// TIA Portal V19 export
FUNCTION_BLOCK "F_Zone01_02_03_FB"   // FB114, F_LAD
TITLE = SAFETY ZONE 01 (DEC.ROTATION) / ZONE 02 (DECOILER 1) / ZONE 03 (DECOILER 2)
// stored: Access Published
   VAR
      D01 : "Door_FB";
      D02 : "Door_FB";
      D03 : "Door_FB";
      F_SafetyValve_DecoilersHorizRotation : "FDevice_Valve_FB";
      F_SafetyValve_Decoiler1 : "FDevice_Valve_FB";
      F_SafetyValve_Decoiler2 : "FDevice_Valve_FB";
      F_Contactor_HU_Decoilers_Motor : "FDevice_Contactor_FB";
      F_Sinamics_DecoilersTranslation : "FDevice_Sinamics_FB";
      F_Sinamics_Decoiler1 : "FDevice_Sinamics_FB";
      F_Sinamics_Decoiler2 : "FDevice_Sinamics_FB";
      Zone02_Close : Bool;
      Zone03_Close : Bool;
   END_VAR
   VAR CONSTANT
      DECOILER_S120_STOPPING_TIME : Time := t#2S;
   END_VAR
BEGIN

REGION Network 1: < < < < < < < < < < DOORS > > > > > > > > > >
END_REGION

REGION Network 2: Zone 01 - Entry enable
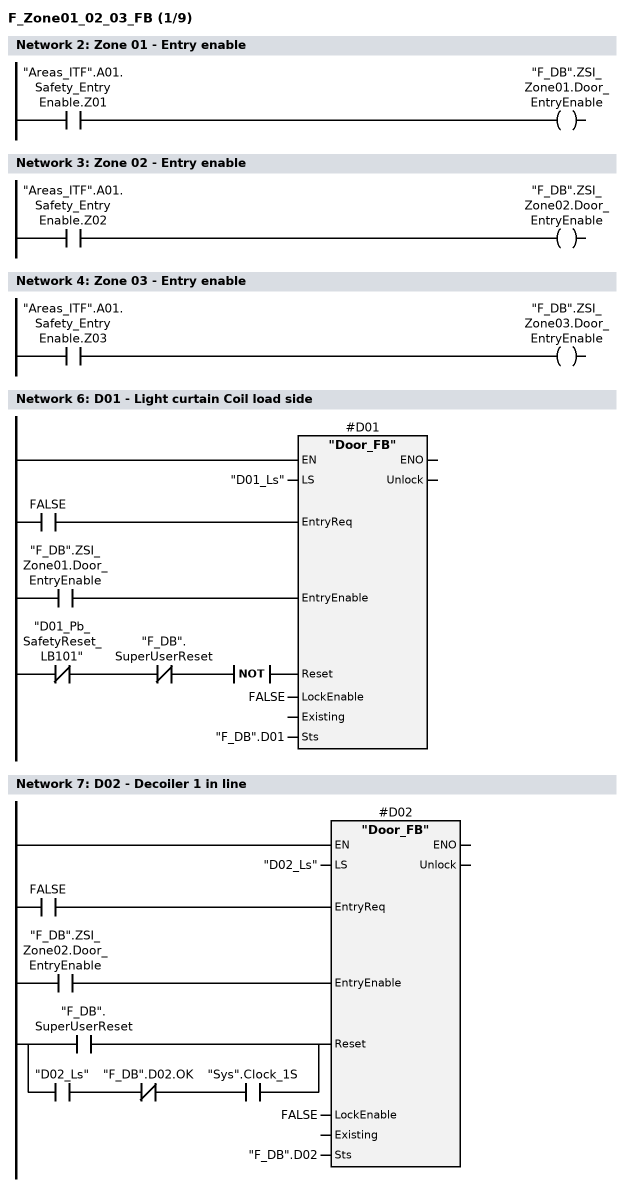
   RUNG wire#powerrail
      Contact( "Areas_ITF".A01.Safety_EntryEnable.Z01 )
      Coil( "F_DB".ZSI_Zone01.Door_EntryEnable )
   END_RUNG
   // the same network as SCL:
   "F_DB".ZSI_Zone01.Door_EntryEnable := "Areas_ITF".A01.Safety_EntryEnable.Z01;
END_REGION

REGION Network 3: Zone 02 - Entry enable
   RUNG wire#powerrail
      Contact( "Areas_ITF".A01.Safety_EntryEnable.Z02 )
      Coil( "F_DB".ZSI_Zone02.Door_EntryEnable )
   END_RUNG
   // the same network as SCL:
   "F_DB".ZSI_Zone02.Door_EntryEnable := "Areas_ITF".A01.Safety_EntryEnable.Z02;
END_REGION

REGION Network 4: Zone 03 - Entry enable
   RUNG wire#powerrail
      Contact( "Areas_ITF".A01.Safety_EntryEnable.Z03 )
      Coil( "F_DB".ZSI_Zone03.Door_EntryEnable )
   END_RUNG
   // the same network as SCL:
   "F_DB".ZSI_Zone03.Door_EntryEnable := "Areas_ITF".A01.Safety_EntryEnable.Z03;
END_REGION

REGION Network 5: >
END_REGION

REGION Network 6: D01 - Light curtain Coil load side
   RUNG wire#powerrail
      #D01(EntryReq := wire#w1, EntryEnable := wire#w2, Reset := wire#w3, LS := "D01_Ls", LockEnable := FALSE, Existing :=, Sts := "F_DB".D01, Unlock =>)
   END_RUNG
   RUNG wire#powerrail
      Contact( FALSE )
   END_RUNG wire#w1
   RUNG wire#powerrail
      Contact( "F_DB".ZSI_Zone01.Door_EntryEnable )
   END_RUNG wire#w2
   RUNG wire#powerrail
      I_Contact( "D01_Pb_SafetyReset_LB101" )
      I_Contact( "F_DB".SuperUserReset )
      Not()
   END_RUNG wire#w3
   // the same network as SCL:
   #D01(LS := "D01_Ls",   // "Door_FB"
        EntryReq := FALSE,
        EntryEnable := "F_DB".ZSI_Zone01.Door_EntryEnable,
        Reset := NOT (NOT "D01_Pb_SafetyReset_LB101" AND NOT "F_DB".SuperUserReset),
        LockEnable := FALSE,
        Sts := "F_DB".D01);
END_REGION

REGION Network 7: D02 - Decoiler 1 in line
   RUNG wire#powerrail
      #D02(EntryReq := wire#w1, EntryEnable := wire#w2, Reset := wire#w3, LS := "D02_Ls", LockEnable := FALSE, Existing :=, Sts := "F_DB".D02, Unlock =>)
   END_RUNG
   RUNG wire#powerrail
      Contact( FALSE )
   END_RUNG wire#w1
   RUNG wire#powerrail
      Contact( "F_DB".ZSI_Zone02.Door_EntryEnable )
   END_RUNG wire#w2
   RUNG wire#powerrail
      Contact( "F_DB".SuperUserReset )
   END_RUNG wire#w3
   RUNG wire#powerrail
      Contact( "D02_Ls" )
      I_Contact( "F_DB".D02.OK )
      Contact( "Sys".Clock_1S )
   END_RUNG wire#w3
   // the same network as SCL:
   #D02(LS := "D02_Ls",   // "Door_FB"
        EntryReq := FALSE,
        EntryEnable := "F_DB".ZSI_Zone02.Door_EntryEnable,
        Reset := "F_DB".SuperUserReset OR ("D02_Ls" AND NOT "F_DB".D02.OK AND "Sys".Clock_1S),
        LockEnable := FALSE,
        Sts := "F_DB".D02);
END_REGION

REGION Network 8: D03 - Decoiler 2 in line
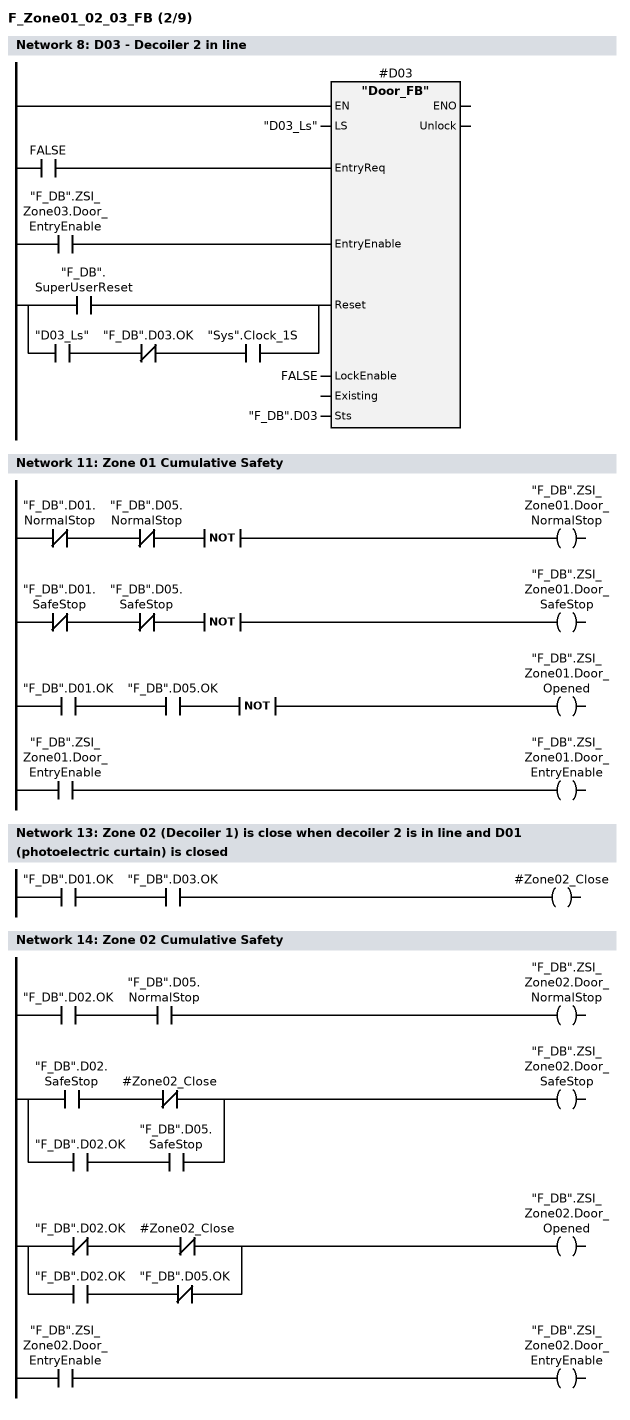
   RUNG wire#powerrail
      #D03(EntryReq := wire#w1, EntryEnable := wire#w2, Reset := wire#w3, LS := "D03_Ls", LockEnable := FALSE, Existing :=, Sts := "F_DB".D03, Unlock =>)
   END_RUNG
   RUNG wire#powerrail
      Contact( FALSE )
   END_RUNG wire#w1
   RUNG wire#powerrail
      Contact( "F_DB".ZSI_Zone03.Door_EntryEnable )
   END_RUNG wire#w2
   RUNG wire#powerrail
      Contact( "F_DB".SuperUserReset )
   END_RUNG wire#w3
   RUNG wire#powerrail
      Contact( "D03_Ls" )
      I_Contact( "F_DB".D03.OK )
      Contact( "Sys".Clock_1S )
   END_RUNG wire#w3
   // the same network as SCL:
   #D03(LS := "D03_Ls",   // "Door_FB"
        EntryReq := FALSE,
        EntryEnable := "F_DB".ZSI_Zone03.Door_EntryEnable,
        Reset := "F_DB".SuperUserReset OR ("D03_Ls" AND NOT "F_DB".D03.OK AND "Sys".Clock_1S),
        LockEnable := FALSE,
        Sts := "F_DB".D03);
END_REGION

REGION Network 9: >
END_REGION

REGION Network 10: < < < < < < < < < < ZONE SAFETY INTERFACE > > > > > > > > > >
END_REGION

REGION Network 11: Zone 01 Cumulative Safety
   RUNG wire#powerrail
      I_Contact( "F_DB".D01.NormalStop )
      I_Contact( "F_DB".D05.NormalStop )
      Not()
      Coil( "F_DB".ZSI_Zone01.Door_NormalStop )
   END_RUNG
   RUNG wire#powerrail
      I_Contact( "F_DB".D01.SafeStop )
      I_Contact( "F_DB".D05.SafeStop )
      Not()
      Coil( "F_DB".ZSI_Zone01.Door_SafeStop )
   END_RUNG
   RUNG wire#powerrail
      Contact( "F_DB".D01.OK )
      Contact( "F_DB".D05.OK )
      Not()
      Coil( "F_DB".ZSI_Zone01.Door_Opened )
   END_RUNG
   RUNG wire#powerrail
      Contact( "F_DB".ZSI_Zone01.Door_EntryEnable )
      Coil( "F_DB".ZSI_Zone01.Door_EntryEnable )
   END_RUNG
   // the same network as SCL:
   "F_DB".ZSI_Zone01.Door_NormalStop := NOT (NOT "F_DB".D01.NormalStop AND NOT "F_DB".D05.NormalStop);
   "F_DB".ZSI_Zone01.Door_SafeStop := NOT (NOT "F_DB".D01.SafeStop AND NOT "F_DB".D05.SafeStop);
   "F_DB".ZSI_Zone01.Door_Opened := NOT ("F_DB".D01.OK AND "F_DB".D05.OK);
   "F_DB".ZSI_Zone01.Door_EntryEnable := "F_DB".ZSI_Zone01.Door_EntryEnable;
END_REGION

REGION Network 12: >
END_REGION

REGION Network 13: Zone 02 (Decoiler 1) is close when decoiler 2 is in line and D01 (photoelectric curtain) is closed
   RUNG wire#powerrail
      Contact( "F_DB".D01.OK )
      Contact( "F_DB".D03.OK )
      Coil( #Zone02_Close )
   END_RUNG
   // the same network as SCL:
   #Zone02_Close := "F_DB".D01.OK AND "F_DB".D03.OK;
END_REGION

REGION Network 14: Zone 02 Cumulative Safety
   RUNG wire#powerrail
      Contact( "F_DB".D02.OK )
      Contact( "F_DB".D05.NormalStop )
      Coil( "F_DB".ZSI_Zone02.Door_NormalStop )
   END_RUNG
   RUNG wire#powerrail
      Contact( "F_DB".D02.SafeStop )
      I_Contact( #Zone02_Close )
      wire#w1
      Coil( "F_DB".ZSI_Zone02.Door_SafeStop )
   END_RUNG
   RUNG wire#powerrail
      Contact( "F_DB".D02.OK )
      Contact( "F_DB".D05.SafeStop )
   END_RUNG wire#w1
   RUNG wire#powerrail
      I_Contact( "F_DB".D02.OK )
      I_Contact( #Zone02_Close )
      wire#w2
      Coil( "F_DB".ZSI_Zone02.Door_Opened )
   END_RUNG
   RUNG wire#powerrail
      Contact( "F_DB".D02.OK )
      I_Contact( "F_DB".D05.OK )
   END_RUNG wire#w2
   RUNG wire#powerrail
      Contact( "F_DB".ZSI_Zone02.Door_EntryEnable )
      Coil( "F_DB".ZSI_Zone02.Door_EntryEnable )
   END_RUNG
   // the same network as SCL:
   "F_DB".ZSI_Zone02.Door_NormalStop := "F_DB".D02.OK AND "F_DB".D05.NormalStop;
   "F_DB".ZSI_Zone02.Door_SafeStop := ("F_DB".D02.SafeStop AND NOT #Zone02_Close) OR ("F_DB".D02.OK AND "F_DB".D05.SafeStop);
   "F_DB".ZSI_Zone02.Door_Opened := (NOT "F_DB".D02.OK AND NOT #Zone02_Close) OR ("F_DB".D02.OK AND NOT "F_DB".D05.OK);
   "F_DB".ZSI_Zone02.Door_EntryEnable := "F_DB".ZSI_Zone02.Door_EntryEnable;
END_REGION

REGION Network 15: >
END_REGION

REGION Network 16: Zone 03 (Decoiler 2) is close when decoiler 1 is in line and D01 (photoelectric curtain) is closed
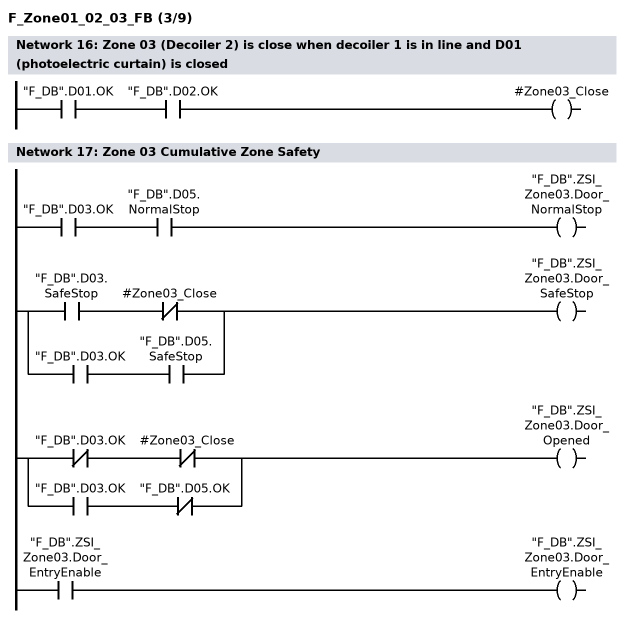
   RUNG wire#powerrail
      Contact( "F_DB".D01.OK )
      Contact( "F_DB".D02.OK )
      Coil( #Zone03_Close )
   END_RUNG
   // the same network as SCL:
   #Zone03_Close := "F_DB".D01.OK AND "F_DB".D02.OK;
END_REGION

REGION Network 17: Zone 03 Cumulative Zone Safety
   RUNG wire#powerrail
      Contact( "F_DB".D03.OK )
      Contact( "F_DB".D05.NormalStop )
      Coil( "F_DB".ZSI_Zone03.Door_NormalStop )
   END_RUNG
   RUNG wire#powerrail
      Contact( "F_DB".D03.SafeStop )
      I_Contact( #Zone03_Close )
      wire#w1
      Coil( "F_DB".ZSI_Zone03.Door_SafeStop )
   END_RUNG
   RUNG wire#powerrail
      Contact( "F_DB".D03.OK )
      Contact( "F_DB".D05.SafeStop )
   END_RUNG wire#w1
   RUNG wire#powerrail
      I_Contact( "F_DB".D03.OK )
      I_Contact( #Zone03_Close )
      wire#w2
      Coil( "F_DB".ZSI_Zone03.Door_Opened )
   END_RUNG
   RUNG wire#powerrail
      Contact( "F_DB".D03.OK )
      I_Contact( "F_DB".D05.OK )
   END_RUNG wire#w2
   RUNG wire#powerrail
      Contact( "F_DB".ZSI_Zone03.Door_EntryEnable )
      Coil( "F_DB".ZSI_Zone03.Door_EntryEnable )
   END_RUNG
   // the same network as SCL:
   "F_DB".ZSI_Zone03.Door_NormalStop := "F_DB".D03.OK AND "F_DB".D05.NormalStop;
   "F_DB".ZSI_Zone03.Door_SafeStop := ("F_DB".D03.SafeStop AND NOT #Zone03_Close) OR ("F_DB".D03.OK AND "F_DB".D05.SafeStop);
   "F_DB".ZSI_Zone03.Door_Opened := (NOT "F_DB".D03.OK AND NOT #Zone03_Close) OR ("F_DB".D03.OK AND NOT "F_DB".D05.OK);
   "F_DB".ZSI_Zone03.Door_EntryEnable := "F_DB".ZSI_Zone03.Door_EntryEnable;
END_REGION

REGION Network 18: >
END_REGION

REGION Network 19: < < < < < < < < < < DEVICES SAFETY VALVES > > > > > > > > > >
END_REGION

REGION Network 20: (Zone 01) HU Decoilers Safety Valve Decoilers Horizonatal Rotation
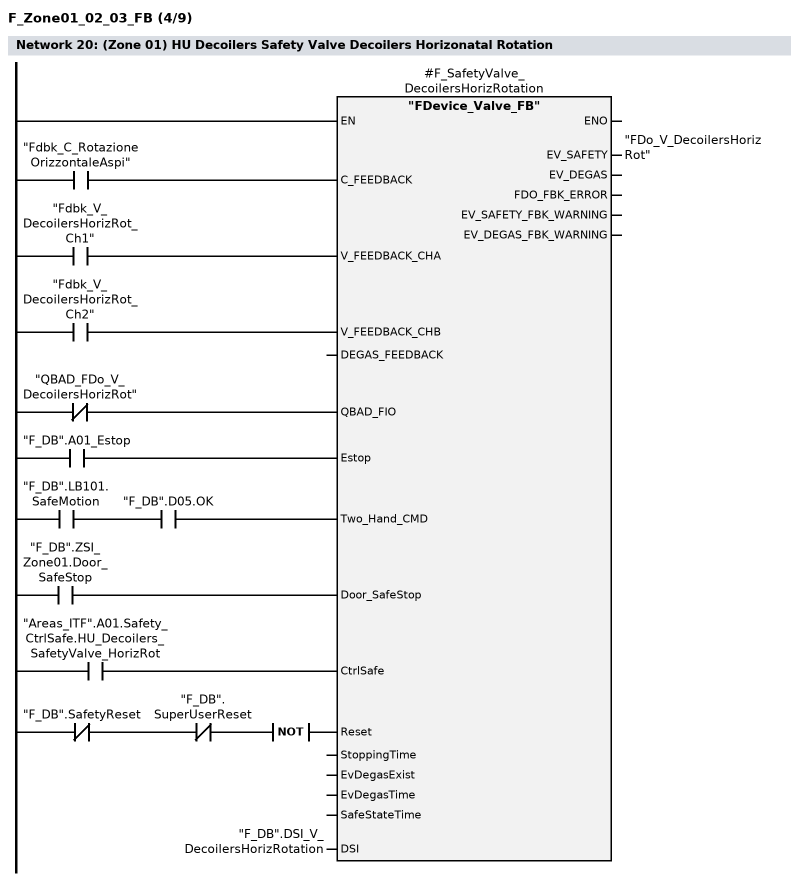
   RUNG wire#powerrail
      #F_SafetyValve_DecoilersHorizRotation(C_FEEDBACK := wire#w1, V_FEEDBACK_CHA := wire#w2, V_FEEDBACK_CHB := wire#w3, QBAD_FIO := wire#w4, Estop := wire#w5, Two_Hand_CMD := wire#w6, Door_SafeStop := wire#w7, CtrlSafe := wire#w8, Reset := wire#w9, DEGAS_FEEDBACK :=, StoppingTime :=, EvDegasExist :=, EvDegasTime :=, SafeStateTime :=, DSI := "F_DB".DSI_V_DecoilersHorizRotation, EV_SAFETY => "FDo_V_DecoilersHorizRot", EV_DEGAS =>, FDO_FBK_ERROR =>, EV_SAFETY_FBK_WARNING =>, EV_DEGAS_FBK_WARNING =>)
   END_RUNG
   RUNG wire#powerrail
      Contact( "Fdbk_C_RotazioneOrizzontaleAspi" )
   END_RUNG wire#w1
   RUNG wire#powerrail
      Contact( "Fdbk_V_DecoilersHorizRot_Ch1" )
   END_RUNG wire#w2
   RUNG wire#powerrail
      Contact( "Fdbk_V_DecoilersHorizRot_Ch2" )
   END_RUNG wire#w3
   RUNG wire#powerrail
      I_Contact( "QBAD_FDo_V_DecoilersHorizRot" )
   END_RUNG wire#w4
   RUNG wire#powerrail
      Contact( "F_DB".A01_Estop )
   END_RUNG wire#w5
   RUNG wire#powerrail
      Contact( "F_DB".LB101.SafeMotion )
      Contact( "F_DB".D05.OK )
   END_RUNG wire#w6
   RUNG wire#powerrail
      Contact( "F_DB".ZSI_Zone01.Door_SafeStop )
   END_RUNG wire#w7
   RUNG wire#powerrail
      Contact( "Areas_ITF".A01.Safety_CtrlSafe.HU_Decoilers_SafetyValve_HorizRot )
   END_RUNG wire#w8
   RUNG wire#powerrail
      I_Contact( "F_DB".SafetyReset )
      I_Contact( "F_DB".SuperUserReset )
      Not()
   END_RUNG wire#w9
   // the same network as SCL:
   #F_SafetyValve_DecoilersHorizRotation(C_FEEDBACK := "Fdbk_C_RotazioneOrizzontaleAspi",   // "FDevice_Valve_FB"
                           V_FEEDBACK_CHA := "Fdbk_V_DecoilersHorizRot_Ch1",
                           V_FEEDBACK_CHB := "Fdbk_V_DecoilersHorizRot_Ch2",
                           QBAD_FIO := NOT "QBAD_FDo_V_DecoilersHorizRot",
                           Estop := "F_DB".A01_Estop,
                           Two_Hand_CMD := "F_DB".LB101.SafeMotion AND "F_DB".D05.OK,
                           Door_SafeStop := "F_DB".ZSI_Zone01.Door_SafeStop,
                           CtrlSafe := "Areas_ITF".A01.Safety_CtrlSafe.HU_Decoilers_SafetyValve_HorizRot,
                           Reset := NOT (NOT "F_DB".SafetyReset AND NOT "F_DB".SuperUserReset),
                           DSI := "F_DB".DSI_V_DecoilersHorizRotation,
                           EV_SAFETY => "FDo_V_DecoilersHorizRot");
END_REGION

REGION Network 21: (Zone 02) HU Decoilers Safety Valve Decoiler 1
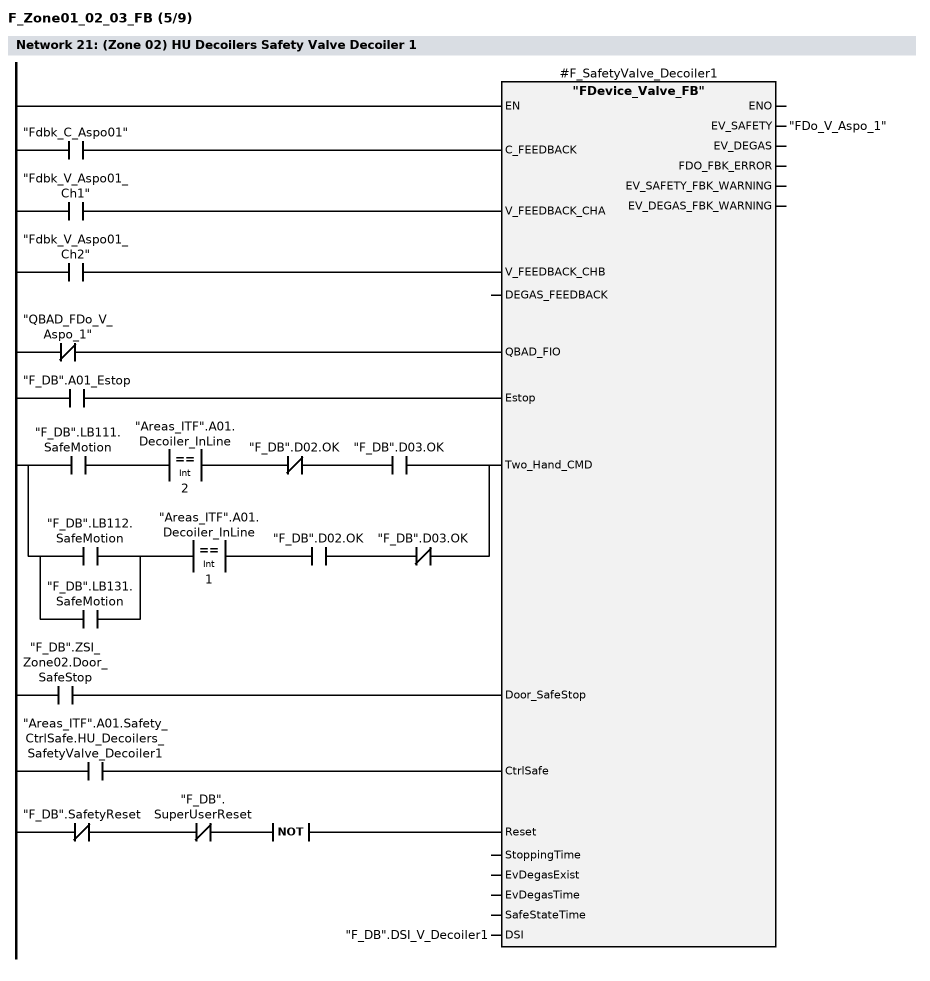
   RUNG wire#powerrail
      #F_SafetyValve_Decoiler1(C_FEEDBACK := wire#w1, V_FEEDBACK_CHA := wire#w2, V_FEEDBACK_CHB := wire#w3, QBAD_FIO := wire#w4, Estop := wire#w5, Two_Hand_CMD := wire#w7, Door_SafeStop := wire#w8, CtrlSafe := wire#w9, Reset := wire#w10, DEGAS_FEEDBACK :=, StoppingTime :=, EvDegasExist :=, EvDegasTime :=, SafeStateTime :=, DSI := "F_DB".DSI_V_Decoiler1, EV_SAFETY => "FDo_V_Aspo_1", EV_DEGAS =>, FDO_FBK_ERROR =>, EV_SAFETY_FBK_WARNING =>, EV_DEGAS_FBK_WARNING =>)
   END_RUNG
   RUNG wire#powerrail
      Contact( "Fdbk_C_Aspo01" )
   END_RUNG wire#w1
   RUNG wire#powerrail
      Contact( "Fdbk_V_Aspo01_Ch1" )
   END_RUNG wire#w2
   RUNG wire#powerrail
      Contact( "Fdbk_V_Aspo01_Ch2" )
   END_RUNG wire#w3
   RUNG wire#powerrail
      I_Contact( "QBAD_FDo_V_Aspo_1" )
   END_RUNG wire#w4
   RUNG wire#powerrail
      Contact( "F_DB".A01_Estop )
   END_RUNG wire#w5
   RUNG wire#powerrail
      Contact( "F_DB".LB111.SafeMotion )
      { S7_Templates := "SrcType := Int" } EQ_Contact(in1 := "Areas_ITF".A01.Decoiler_InLine, in2 := 2)
      I_Contact( "F_DB".D02.OK )
      Contact( "F_DB".D03.OK )
   END_RUNG wire#w7
   RUNG wire#powerrail
      Contact( "F_DB".LB112.SafeMotion )
      wire#w6
      { S7_Templates := "SrcType := Int" } EQ_Contact(in1 := "Areas_ITF".A01.Decoiler_InLine, in2 := 1)
      Contact( "F_DB".D02.OK )
      I_Contact( "F_DB".D03.OK )
   END_RUNG wire#w7
   RUNG wire#powerrail
      Contact( "F_DB".LB131.SafeMotion )
   END_RUNG wire#w6
   RUNG wire#powerrail
      Contact( "F_DB".ZSI_Zone02.Door_SafeStop )
   END_RUNG wire#w8
   RUNG wire#powerrail
      Contact( "Areas_ITF".A01.Safety_CtrlSafe.HU_Decoilers_SafetyValve_Decoiler1 )
   END_RUNG wire#w9
   RUNG wire#powerrail
      I_Contact( "F_DB".SafetyReset )
      I_Contact( "F_DB".SuperUserReset )
      Not()
   END_RUNG wire#w10
   // the same network as SCL:
   #F_SafetyValve_Decoiler1(C_FEEDBACK := "Fdbk_C_Aspo01",   // "FDevice_Valve_FB"
                           V_FEEDBACK_CHA := "Fdbk_V_Aspo01_Ch1",
                           V_FEEDBACK_CHB := "Fdbk_V_Aspo01_Ch2",
                           QBAD_FIO := NOT "QBAD_FDo_V_Aspo_1",
                           Estop := "F_DB".A01_Estop,
                           Two_Hand_CMD := ("F_DB".LB111.SafeMotion AND ("Areas_ITF".A01.Decoiler_InLine = 2) AND NOT "F_DB".D02.OK AND "F_DB".D03.OK) OR (("F_DB".LB112.SafeMotion OR "F_DB".LB131.SafeMotion) AND ("Areas_ITF".A01.Decoiler_InLine = 1) AND "F_DB".D02.OK AND NOT "F_DB".D03.OK),
                           Door_SafeStop := "F_DB".ZSI_Zone02.Door_SafeStop,
                           CtrlSafe := "Areas_ITF".A01.Safety_CtrlSafe.HU_Decoilers_SafetyValve_Decoiler1,
                           Reset := NOT (NOT "F_DB".SafetyReset AND NOT "F_DB".SuperUserReset),
                           DSI := "F_DB".DSI_V_Decoiler1,
                           EV_SAFETY => "FDo_V_Aspo_1");
END_REGION

REGION Network 22: (Zone 03) HU Decoilers Safety Valve Decoiler 2
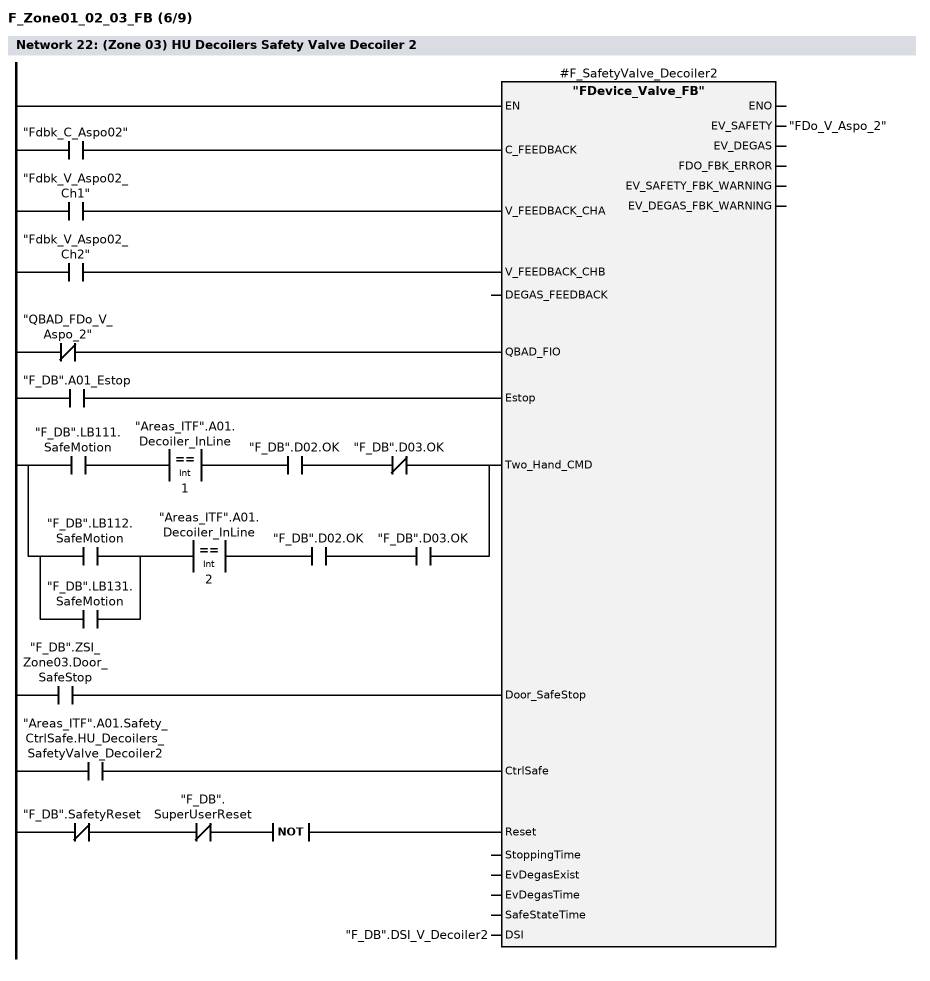
   RUNG wire#powerrail
      #F_SafetyValve_Decoiler2(C_FEEDBACK := wire#w1, V_FEEDBACK_CHA := wire#w2, V_FEEDBACK_CHB := wire#w3, QBAD_FIO := wire#w4, Estop := wire#w5, Two_Hand_CMD := wire#w7, Door_SafeStop := wire#w8, CtrlSafe := wire#w9, Reset := wire#w10, DEGAS_FEEDBACK :=, StoppingTime :=, EvDegasExist :=, EvDegasTime :=, SafeStateTime :=, DSI := "F_DB".DSI_V_Decoiler2, EV_SAFETY => "FDo_V_Aspo_2", EV_DEGAS =>, FDO_FBK_ERROR =>, EV_SAFETY_FBK_WARNING =>, EV_DEGAS_FBK_WARNING =>)
   END_RUNG
   RUNG wire#powerrail
      Contact( "Fdbk_C_Aspo02" )
   END_RUNG wire#w1
   RUNG wire#powerrail
      Contact( "Fdbk_V_Aspo02_Ch1" )
   END_RUNG wire#w2
   RUNG wire#powerrail
      Contact( "Fdbk_V_Aspo02_Ch2" )
   END_RUNG wire#w3
   RUNG wire#powerrail
      I_Contact( "QBAD_FDo_V_Aspo_2" )
   END_RUNG wire#w4
   RUNG wire#powerrail
      Contact( "F_DB".A01_Estop )
   END_RUNG wire#w5
   RUNG wire#powerrail
      Contact( "F_DB".LB111.SafeMotion )
      { S7_Templates := "SrcType := Int" } EQ_Contact(in1 := "Areas_ITF".A01.Decoiler_InLine, in2 := 1)
      Contact( "F_DB".D02.OK )
      I_Contact( "F_DB".D03.OK )
   END_RUNG wire#w7
   RUNG wire#powerrail
      Contact( "F_DB".LB112.SafeMotion )
      wire#w6
      { S7_Templates := "SrcType := Int" } EQ_Contact(in1 := "Areas_ITF".A01.Decoiler_InLine, in2 := 2)
      Contact( "F_DB".D02.OK )
      Contact( "F_DB".D03.OK )
   END_RUNG wire#w7
   RUNG wire#powerrail
      Contact( "F_DB".LB131.SafeMotion )
   END_RUNG wire#w6
   RUNG wire#powerrail
      Contact( "F_DB".ZSI_Zone03.Door_SafeStop )
   END_RUNG wire#w8
   RUNG wire#powerrail
      Contact( "Areas_ITF".A01.Safety_CtrlSafe.HU_Decoilers_SafetyValve_Decoiler2 )
   END_RUNG wire#w9
   RUNG wire#powerrail
      I_Contact( "F_DB".SafetyReset )
      I_Contact( "F_DB".SuperUserReset )
      Not()
   END_RUNG wire#w10
   // the same network as SCL:
   #F_SafetyValve_Decoiler2(C_FEEDBACK := "Fdbk_C_Aspo02",   // "FDevice_Valve_FB"
                           V_FEEDBACK_CHA := "Fdbk_V_Aspo02_Ch1",
                           V_FEEDBACK_CHB := "Fdbk_V_Aspo02_Ch2",
                           QBAD_FIO := NOT "QBAD_FDo_V_Aspo_2",
                           Estop := "F_DB".A01_Estop,
                           Two_Hand_CMD := ("F_DB".LB111.SafeMotion AND ("Areas_ITF".A01.Decoiler_InLine = 1) AND "F_DB".D02.OK AND NOT "F_DB".D03.OK) OR (("F_DB".LB112.SafeMotion OR "F_DB".LB131.SafeMotion) AND ("Areas_ITF".A01.Decoiler_InLine = 2) AND "F_DB".D02.OK AND "F_DB".D03.OK),
                           Door_SafeStop := "F_DB".ZSI_Zone03.Door_SafeStop,
                           CtrlSafe := "Areas_ITF".A01.Safety_CtrlSafe.HU_Decoilers_SafetyValve_Decoiler2,
                           Reset := NOT (NOT "F_DB".SafetyReset AND NOT "F_DB".SuperUserReset),
                           DSI := "F_DB".DSI_V_Decoiler2,
                           EV_SAFETY => "FDo_V_Aspo_2");
END_REGION

REGION Network 23: >
END_REGION

REGION Network 24: < < < < < < < < < < DEVICES CONTACTORS > > > > > > > > > >
END_REGION

REGION Network 25: (Zone 01-02-03) HU Decoiler Motor contactor
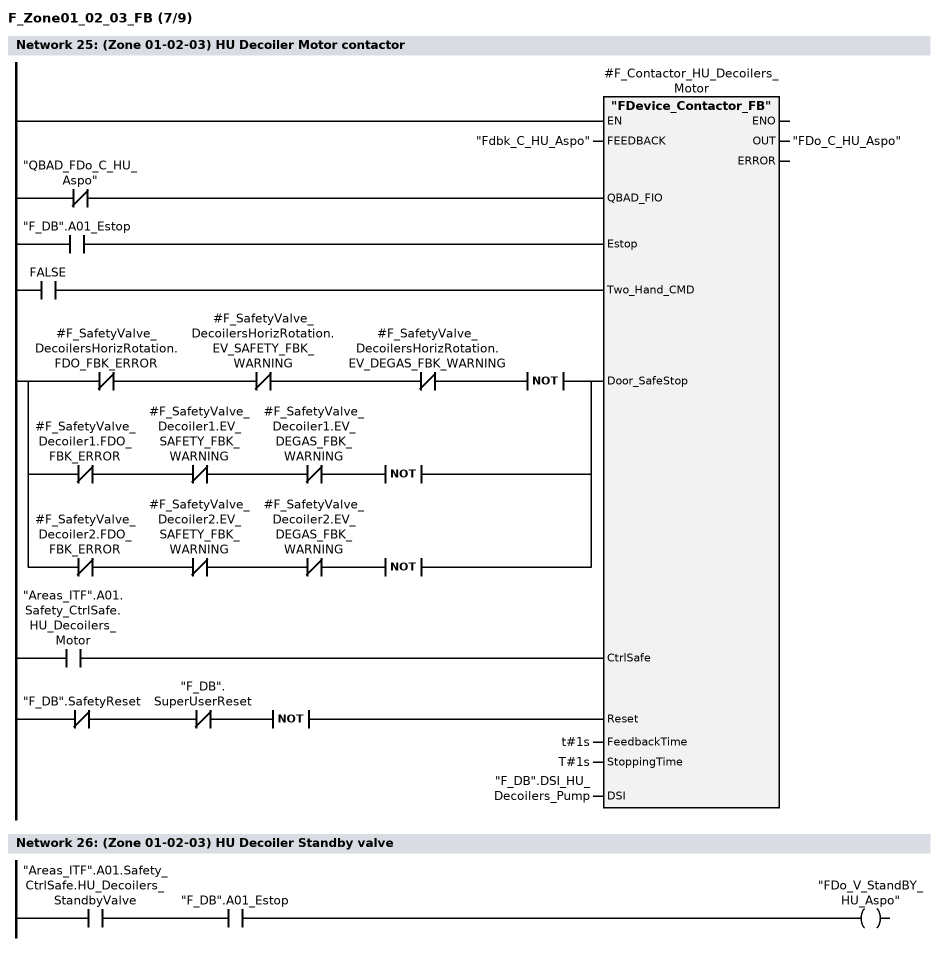
   RUNG wire#powerrail
      #F_Contactor_HU_Decoilers_Motor(QBAD_FIO := wire#w1, Estop := wire#w2, Two_Hand_CMD := wire#w3, Door_SafeStop := wire#w4, CtrlSafe := wire#w5, Reset := wire#w6, FEEDBACK := "Fdbk_C_HU_Aspo", FeedbackTime := t#1s, StoppingTime := T#1s, DSI := "F_DB".DSI_HU_Decoilers_Pump, OUT => "FDo_C_HU_Aspo", ERROR =>)
   END_RUNG
   RUNG wire#powerrail
      I_Contact( "QBAD_FDo_C_HU_Aspo" )
   END_RUNG wire#w1
   RUNG wire#powerrail
      Contact( "F_DB".A01_Estop )
   END_RUNG wire#w2
   RUNG wire#powerrail
      Contact( FALSE )
   END_RUNG wire#w3
   RUNG wire#powerrail
      I_Contact( #F_SafetyValve_DecoilersHorizRotation.FDO_FBK_ERROR )
      I_Contact( #F_SafetyValve_DecoilersHorizRotation.EV_SAFETY_FBK_WARNING )
      I_Contact( #F_SafetyValve_DecoilersHorizRotation.EV_DEGAS_FBK_WARNING )
      Not()
   END_RUNG wire#w4
   RUNG wire#powerrail
      I_Contact( #F_SafetyValve_Decoiler1.FDO_FBK_ERROR )
      I_Contact( #F_SafetyValve_Decoiler1.EV_SAFETY_FBK_WARNING )
      I_Contact( #F_SafetyValve_Decoiler1.EV_DEGAS_FBK_WARNING )
      Not()
   END_RUNG wire#w4
   RUNG wire#powerrail
      I_Contact( #F_SafetyValve_Decoiler2.FDO_FBK_ERROR )
      I_Contact( #F_SafetyValve_Decoiler2.EV_SAFETY_FBK_WARNING )
      I_Contact( #F_SafetyValve_Decoiler2.EV_DEGAS_FBK_WARNING )
      Not()
   END_RUNG wire#w4
   RUNG wire#powerrail
      Contact( "Areas_ITF".A01.Safety_CtrlSafe.HU_Decoilers_Motor )
   END_RUNG wire#w5
   RUNG wire#powerrail
      I_Contact( "F_DB".SafetyReset )
      I_Contact( "F_DB".SuperUserReset )
      Not()
   END_RUNG wire#w6
   // the same network as SCL:
   #F_Contactor_HU_Decoilers_Motor(FEEDBACK := "Fdbk_C_HU_Aspo",   // "FDevice_Contactor_FB"
                           QBAD_FIO := NOT "QBAD_FDo_C_HU_Aspo",
                           Estop := "F_DB".A01_Estop,
                           Two_Hand_CMD := FALSE,
                           Door_SafeStop := NOT (NOT #F_SafetyValve_DecoilersHorizRotation.FDO_FBK_ERROR AND NOT #F_SafetyValve_DecoilersHorizRotation.EV_SAFETY_FBK_WARNING AND NOT #F_SafetyValve_DecoilersHorizRotation.EV_DEGAS_FBK_WARNING) OR NOT (NOT #F_SafetyValve_Decoiler1.FDO_FBK_ERROR AND NOT #F_SafetyValve_Decoiler1.EV_SAFETY_FBK_WARNING AND NOT #F_SafetyValve_Decoiler1.EV_DEGAS_FBK_WARNING) OR NOT (NOT #F_SafetyValve_Decoiler2.FDO_FBK_ERROR AND NOT #F_SafetyValve_Decoiler2.EV_SAFETY_FBK_WARNING AND NOT #F_SafetyValve_Decoiler2.EV_DEGAS_FBK_WARNING),
                           CtrlSafe := "Areas_ITF".A01.Safety_CtrlSafe.HU_Decoilers_Motor,
                           Reset := NOT (NOT "F_DB".SafetyReset AND NOT "F_DB".SuperUserReset),
                           FeedbackTime := t#1s,
                           StoppingTime := T#1s,
                           DSI := "F_DB".DSI_HU_Decoilers_Pump,
                           OUT => "FDo_C_HU_Aspo");
END_REGION

REGION Network 26: (Zone 01-02-03) HU Decoiler Standby valve
   RUNG wire#powerrail
      Contact( "Areas_ITF".A01.Safety_CtrlSafe.HU_Decoilers_StandbyValve )
      Contact( "F_DB".A01_Estop )
      Coil( "FDo_V_StandBY_HU_Aspo" )
   END_RUNG
   // the same network as SCL:
   "FDo_V_StandBY_HU_Aspo" := "Areas_ITF".A01.Safety_CtrlSafe.HU_Decoilers_StandbyValve AND "F_DB".A01_Estop;
END_REGION

REGION Network 27: >
END_REGION

REGION Network 28: < < < < < < < < < < DEVICES S120 > > > > > > > > > >
END_REGION

REGION Network 29: (Zone 01) S120 - Decoilers Translation
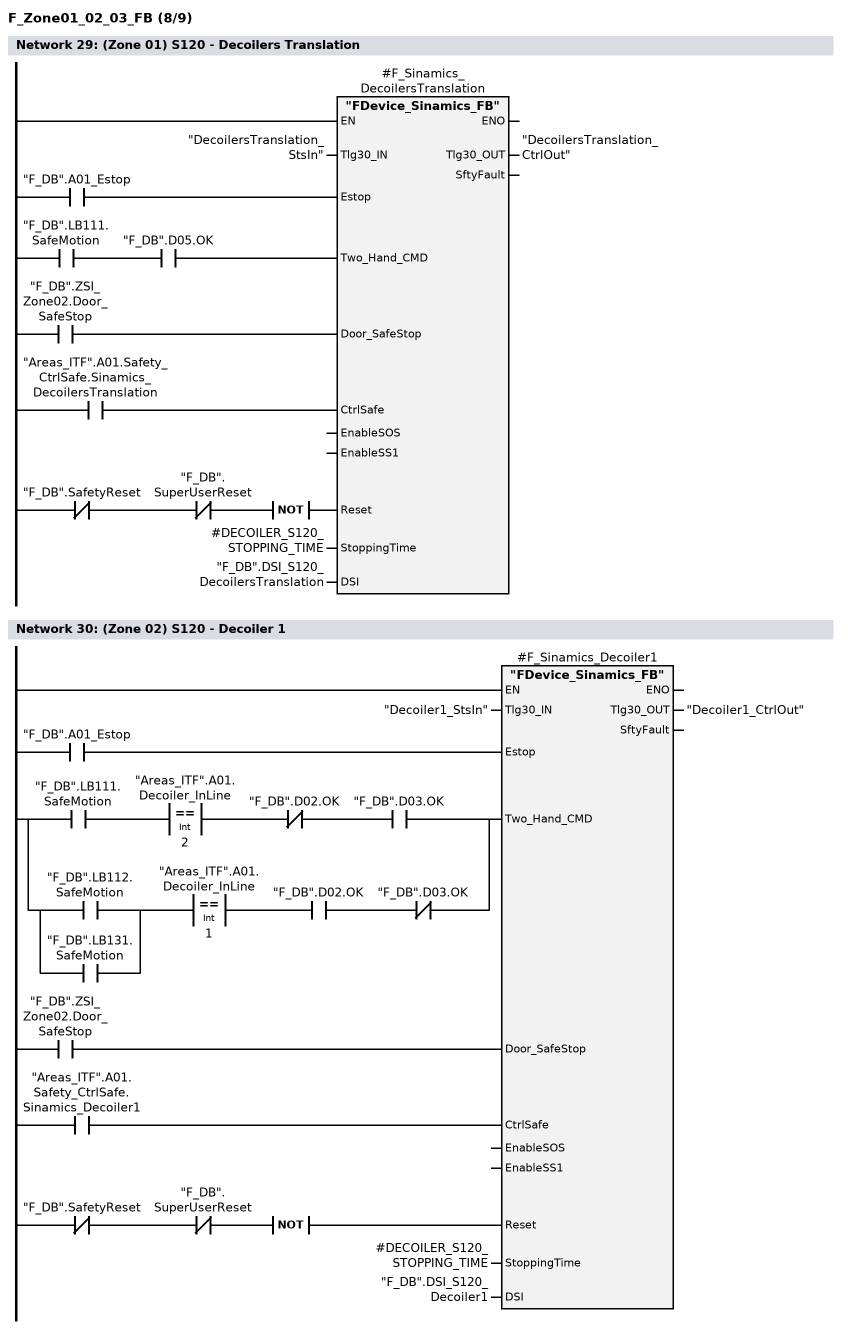
   RUNG wire#powerrail
      #F_Sinamics_DecoilersTranslation(Estop := wire#w1, Two_Hand_CMD := wire#w2, Door_SafeStop := wire#w3, CtrlSafe := wire#w4, Reset := wire#w5, Tlg30_IN := "DecoilersTranslation_StsIn", EnableSOS :=, EnableSS1 :=, StoppingTime := #DECOILER_S120_STOPPING_TIME, DSI := "F_DB".DSI_S120_DecoilersTranslation, Tlg30_OUT => "DecoilersTranslation_CtrlOut", SftyFault =>)
   END_RUNG
   RUNG wire#powerrail
      Contact( "F_DB".A01_Estop )
   END_RUNG wire#w1
   RUNG wire#powerrail
      Contact( "F_DB".LB111.SafeMotion )
      Contact( "F_DB".D05.OK )
   END_RUNG wire#w2
   RUNG wire#powerrail
      Contact( "F_DB".ZSI_Zone02.Door_SafeStop )
   END_RUNG wire#w3
   RUNG wire#powerrail
      Contact( "Areas_ITF".A01.Safety_CtrlSafe.Sinamics_DecoilersTranslation )
   END_RUNG wire#w4
   RUNG wire#powerrail
      I_Contact( "F_DB".SafetyReset )
      I_Contact( "F_DB".SuperUserReset )
      Not()
   END_RUNG wire#w5
   // the same network as SCL:
   #F_Sinamics_DecoilersTranslation(Tlg30_IN := "DecoilersTranslation_StsIn",   // "FDevice_Sinamics_FB"
                           Estop := "F_DB".A01_Estop,
                           Two_Hand_CMD := "F_DB".LB111.SafeMotion AND "F_DB".D05.OK,
                           Door_SafeStop := "F_DB".ZSI_Zone02.Door_SafeStop,
                           CtrlSafe := "Areas_ITF".A01.Safety_CtrlSafe.Sinamics_DecoilersTranslation,
                           Reset := NOT (NOT "F_DB".SafetyReset AND NOT "F_DB".SuperUserReset),
                           StoppingTime := #DECOILER_S120_STOPPING_TIME,
                           DSI := "F_DB".DSI_S120_DecoilersTranslation,
                           Tlg30_OUT => "DecoilersTranslation_CtrlOut");
END_REGION

REGION Network 30: (Zone 02) S120 - Decoiler 1
   RUNG wire#powerrail
      #F_Sinamics_Decoiler1(Estop := wire#w1, Two_Hand_CMD := wire#w3, Door_SafeStop := wire#w4, CtrlSafe := wire#w5, Reset := wire#w6, Tlg30_IN := "Decoiler1_StsIn", EnableSOS :=, EnableSS1 :=, StoppingTime := #DECOILER_S120_STOPPING_TIME, DSI := "F_DB".DSI_S120_Decoiler1, Tlg30_OUT => "Decoiler1_CtrlOut", SftyFault =>)
   END_RUNG
   RUNG wire#powerrail
      Contact( "F_DB".A01_Estop )
   END_RUNG wire#w1
   RUNG wire#powerrail
      Contact( "F_DB".LB111.SafeMotion )
      { S7_Templates := "SrcType := Int" } EQ_Contact(in1 := "Areas_ITF".A01.Decoiler_InLine, in2 := 2)
      I_Contact( "F_DB".D02.OK )
      Contact( "F_DB".D03.OK )
   END_RUNG wire#w3
   RUNG wire#powerrail
      Contact( "F_DB".LB112.SafeMotion )
      wire#w2
      { S7_Templates := "SrcType := Int" } EQ_Contact(in1 := "Areas_ITF".A01.Decoiler_InLine, in2 := 1)
      Contact( "F_DB".D02.OK )
      I_Contact( "F_DB".D03.OK )
   END_RUNG wire#w3
   RUNG wire#powerrail
      Contact( "F_DB".LB131.SafeMotion )
   END_RUNG wire#w2
   RUNG wire#powerrail
      Contact( "F_DB".ZSI_Zone02.Door_SafeStop )
   END_RUNG wire#w4
   RUNG wire#powerrail
      Contact( "Areas_ITF".A01.Safety_CtrlSafe.Sinamics_Decoiler1 )
   END_RUNG wire#w5
   RUNG wire#powerrail
      I_Contact( "F_DB".SafetyReset )
      I_Contact( "F_DB".SuperUserReset )
      Not()
   END_RUNG wire#w6
   // the same network as SCL:
   #F_Sinamics_Decoiler1(Tlg30_IN := "Decoiler1_StsIn",   // "FDevice_Sinamics_FB"
                         Estop := "F_DB".A01_Estop,
                         Two_Hand_CMD := ("F_DB".LB111.SafeMotion AND ("Areas_ITF".A01.Decoiler_InLine = 2) AND NOT "F_DB".D02.OK AND "F_DB".D03.OK) OR (("F_DB".LB112.SafeMotion OR "F_DB".LB131.SafeMotion) AND ("Areas_ITF".A01.Decoiler_InLine = 1) AND "F_DB".D02.OK AND NOT "F_DB".D03.OK),
                         Door_SafeStop := "F_DB".ZSI_Zone02.Door_SafeStop,
                         CtrlSafe := "Areas_ITF".A01.Safety_CtrlSafe.Sinamics_Decoiler1,
                         Reset := NOT (NOT "F_DB".SafetyReset AND NOT "F_DB".SuperUserReset),
                         StoppingTime := #DECOILER_S120_STOPPING_TIME,
                         DSI := "F_DB".DSI_S120_Decoiler1,
                         Tlg30_OUT => "Decoiler1_CtrlOut");
END_REGION

REGION Network 31: (Zone 03) S120 - Decoiler 2
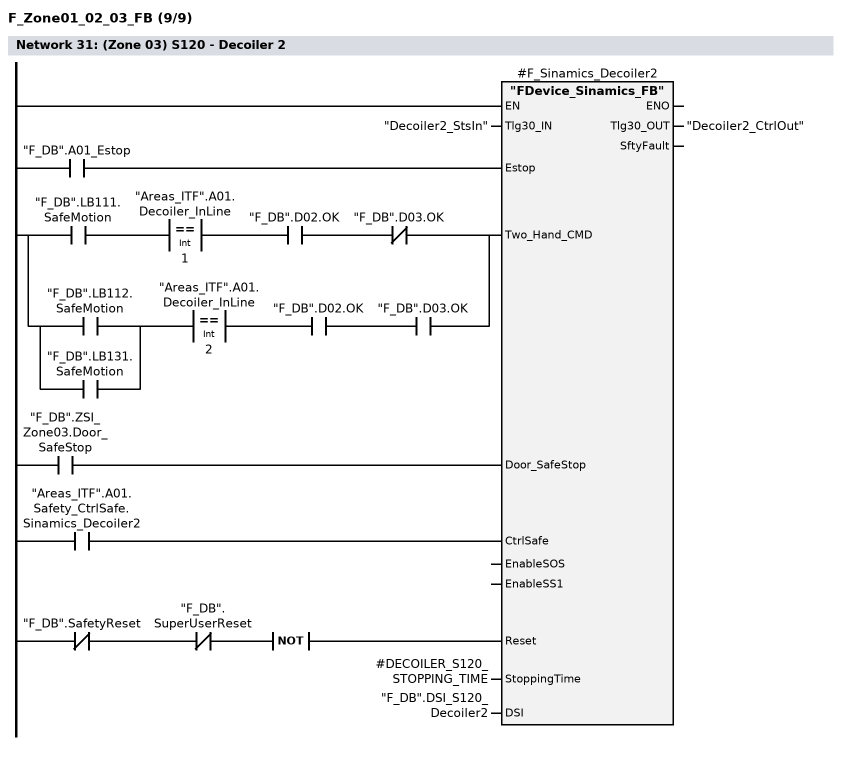
   RUNG wire#powerrail
      #F_Sinamics_Decoiler2(Estop := wire#w1, Two_Hand_CMD := wire#w3, Door_SafeStop := wire#w4, CtrlSafe := wire#w5, Reset := wire#w6, Tlg30_IN := "Decoiler2_StsIn", EnableSOS :=, EnableSS1 :=, StoppingTime := #DECOILER_S120_STOPPING_TIME, DSI := "F_DB".DSI_S120_Decoiler2, Tlg30_OUT => "Decoiler2_CtrlOut", SftyFault =>)
   END_RUNG
   RUNG wire#powerrail
      Contact( "F_DB".A01_Estop )
   END_RUNG wire#w1
   RUNG wire#powerrail
      Contact( "F_DB".LB111.SafeMotion )
      { S7_Templates := "SrcType := Int" } EQ_Contact(in1 := "Areas_ITF".A01.Decoiler_InLine, in2 := 1)
      Contact( "F_DB".D02.OK )
      I_Contact( "F_DB".D03.OK )
   END_RUNG wire#w3
   RUNG wire#powerrail
      Contact( "F_DB".LB112.SafeMotion )
      wire#w2
      { S7_Templates := "SrcType := Int" } EQ_Contact(in1 := "Areas_ITF".A01.Decoiler_InLine, in2 := 2)
      Contact( "F_DB".D02.OK )
      Contact( "F_DB".D03.OK )
   END_RUNG wire#w3
   RUNG wire#powerrail
      Contact( "F_DB".LB131.SafeMotion )
   END_RUNG wire#w2
   RUNG wire#powerrail
      Contact( "F_DB".ZSI_Zone03.Door_SafeStop )
   END_RUNG wire#w4
   RUNG wire#powerrail
      Contact( "Areas_ITF".A01.Safety_CtrlSafe.Sinamics_Decoiler2 )
   END_RUNG wire#w5
   RUNG wire#powerrail
      I_Contact( "F_DB".SafetyReset )
      I_Contact( "F_DB".SuperUserReset )
      Not()
   END_RUNG wire#w6
   // the same network as SCL:
   #F_Sinamics_Decoiler2(Tlg30_IN := "Decoiler2_StsIn",   // "FDevice_Sinamics_FB"
                         Estop := "F_DB".A01_Estop,
                         Two_Hand_CMD := ("F_DB".LB111.SafeMotion AND ("Areas_ITF".A01.Decoiler_InLine = 1) AND "F_DB".D02.OK AND NOT "F_DB".D03.OK) OR (("F_DB".LB112.SafeMotion OR "F_DB".LB131.SafeMotion) AND ("Areas_ITF".A01.Decoiler_InLine = 2) AND "F_DB".D02.OK AND "F_DB".D03.OK),
                         Door_SafeStop := "F_DB".ZSI_Zone03.Door_SafeStop,
                         CtrlSafe := "Areas_ITF".A01.Safety_CtrlSafe.Sinamics_Decoiler2,
                         Reset := NOT (NOT "F_DB".SafetyReset AND NOT "F_DB".SuperUserReset),
                         StoppingTime := #DECOILER_S120_STOPPING_TIME,
                         DSI := "F_DB".DSI_S120_Decoiler2,
                         Tlg30_OUT => "Decoiler2_CtrlOut");
END_REGION

REGION Network 32: >
END_REGION

REGION Network 33: >
END_REGION

REGION Network 34: >
END_REGION
END_FUNCTION_BLOCK
